Staubli VAL3: select.pgx

program select(num& x_nSelect[])
  local num i
  local num l_nIndex
  local num l_nMin
begin
  //
  // to save:
  // x_nBest [0] -# Traejctory
  // x_nBest [1] -# index
  //
  // STRATEGY look the FIRST VALUE
  if nDistance>saveData:nRadiusHome
    // take the first
    l_nIndex=0
  else
    // look for the point beyond the radius
    l_nMin=100000
    for i=0 to size(nDistance)-1
      if nDistance[i]<saveData:nRadiusHome
        if nCoeff[i]<l_nMin and abs(nCoeff[i]-l_nMin)>30
          l_nMin=nCoeff[i]
          l_nIndex=i
          if saveData:bDebug
            ? "searching inside"
            ? nDistance[i]
            ? nJoint[i]
            ? nHome[i]
          endIf
        endIf
      else
        // exit
        i=size(nDistance)-1
      endIf
    endFor
  endIf
  // save the value
  x_nSelect[0]=nHome[l_nIndex]
  x_nSelect[1]=nJoint[l_nIndex]
end
